// TIA Portal V21 export
TYPE "lubricationSystemCmd"
   STRUCT
      oilPump1Selected : Bool;
      oilPump2Selected : Bool;
      cmdWord : Word;
   END_STRUCT;
END_TYPE
